(* PLC project Generated.project, CODESYS CODESYS V3.5 SP19 Patch 1 *)
(* stored: creationDateTime 2026-08-11T14:02:33.677683, modificationDateTime 2026-08-11T14:02:33.677683 *)

(* ═══════════════════════════════════════════════════════════════ 🚦 ST_DredgingAssistState — États publics assistance prélèvement ═══════════════════════════════════════════════════════════════ *)
TYPE ST_DredgingAssistState : STRUCT
  DiveReady : BOOL;
  DiveBusy : BOOL;
  DiveDone : BOOL;
  DiveError : BOOL;
  DiveErrorId : WORD;
  DiveState : E_DiveSearchState;
  BottomTouchConfirmed : BOOL;
  ExtractionReady : BOOL;
  ExtractionBusy : BOOL;
  ExtractionDone : BOOL;
  ExtractionError : BOOL;
  ExtractionErrorId : WORD;
  ExtractionState : E_ExtractionSequenceState;
  OperatorActionId : WORD;  (* Une seule consigne conduite, arbitré en PRG_09 *)
  OperatorAction : STRING(120);  (* Texte de secours ; IHM peut mapper l'identifiant *)
  DumpAtTremieArmed : BOOL;  (* 🆕 2026-08-07 : mode vidage à la trémie (pas de FB dédié, logique combinatoire PRG_04) TglEnableDumpAtTremie (bit IHM brut) *)
  DumpAtTremieAssistActive : BOOL;  (* Armé ET Mode MAINT_N1/N2 (mode réellement actif) *)
  DumpAtTremieAtTremie : BOOL;  (* M3_AtTremieStable *)
  DumpAtTremieBucketOpenArmed : BOOL;  (* CmdOpen_IHM déclenché par ce mode *)
  DumpAtTremieDescentLocked : BOOL;  (* ForbidDescent M1/M2 forcé par ce mode (hors P1/Maintenance) *)
  BypassDiveActive : BOOL;  (* 🆕 2026-08-07 (9) : diagnostic bypass séquence DiveSearch TglBypassDiveSearchSequence armé (descente couplée en cours) *)
  BypassKoboldBottomTouched : BOOL;  (* Fond confirmé par le bypass (front montant Kobold en descente) *)
END_STRUCT;
END_TYPE

(* values of E_DiveSearchState: WAIT_PRECONDITIONS: Attente benne ouverte, positions et Kobold au repos; READY_TO_DESCEND: Prêt à assister une demande de descente; SEARCHING_IMMERSION: Descente : attente front 0→1 dans fenêtre eau; SEARCHING_BOTTOM: Immersion validée : attente front 1→0 au fond; BOTTOM_CONFIRMED: Fond validé ; extraction peut être demandée; ERROR_HOLD: Séquence invalide, descente assistée interdite *)

{attribute 'qualified_only'}
{attribute 'strict'}
TYPE E_DiveSearchState : (WAIT_PRECONDITIONS := 0, READY_TO_DESCEND := 1, SEARCHING_IMMERSION := 2, SEARCHING_BOTTOM := 3, BOTTOM_CONFIRMED := 4, ERROR_HOLD := 5);
END_TYPE

(* values of E_ExtractionSequenceState: WAIT_BOTTOM_CONFIRMATION: Attente fond Kobold ou attestation opérateur; READY_TO_CLOSE: Prêt à fermer la benne; CLOSING_BUCKET: FB_Bucket ferme M2 seul; CONTROL_ASCENT: M1/M2 synchronisés au palier sans contacteur vitesse; NOMINAL_ASCENT: Montée couplée avec vitesse demandée opérateur; ERROR_HOLD: Défaut extraction, reprise interdite avant reset *)

{attribute 'qualified_only'}
{attribute 'strict'}
TYPE E_ExtractionSequenceState : (WAIT_BOTTOM_CONFIRMATION := 0, READY_TO_CLOSE := 1, CLOSING_BUCKET := 2, CONTROL_ASCENT := 3, NOMINAL_ASCENT := 4, ERROR_HOLD := 5);
END_TYPE
